{attribute 'linkalways'} 
{attribute 'no_explicit_call' := 'This FB is a CLASS and must be accessed using methods or properties'}
{attribute 'enable_dynamic_creation'}
FUNCTION_BLOCK Node_F_VN_TransformIntoDisplayableImageExp EXTENDS VisionNode
VAR
    ipSrcImage : _ITcVnImage;
    ipDestImage : _ITcVnDisplayableImage;
    bAllowDeepCopy : _BOOL(FALSE);
    hrPrev : _HRESULT(S_OK);
	hresult : _HRESULT(S_OK);
END_VAR

METHOD PUBLIC  Clone : I_Node
VAR
	pNode : POINTER TO Node_F_VN_TransformIntoDisplayableImageExp;
END_VAR
pNode := __NEW(Node_F_VN_TransformIntoDisplayableImageExp);
Clone := pNode^;
END_METHOD

METHOD FB_init : BOOL
VAR_INPUT
	bInitRetains : BOOL; // if TRUE, the retain variables are initialized (warm start / cold start)
	bInCopyCode : BOOL;  // if TRUE, the instance afterwards gets moved into the copy code (online change)
END_VAR
AddInput('ipSrcImage', ipSrcImage);
AddParameter('bAllowDeepCopy', bAllowDeepCopy);
AddInput('hrPrev', hrPrev);
AddOutput('ipDestImage', ipDestImage);
AddOutput('hresult',hresult);
END_METHOD

METHOD PROTECTED OnExecute
hresult.Value := F_VN_TransformIntoDisplayableImageExp(
    ipSrcImage := ipSrcImage.Value,
    bAllowDeepCopy := bAllowDeepCopy.Value,
	ipDestImage := ipDestImage.Value,
	hrPrev:= hrPrev.Value);
END_METHOD

METHOD PUBLIC PreExecutionCheck
VAR_INPUT
	Check : I_PreExecutionChecks;
END_VAR
Check.IsTrue(ipSrcImage.IsValid, 'ipSrcImage must contain an image');
END_METHOD

END_FUNCTION_BLOCK

(* stored: Version 1.1.0.1, ProductVersion 3.1.4024.15
   POU Node_F_VN_TransformIntoDisplayableImageExp: Id {d1cda9be-a710-05ca-1817-66ea43c7cedf}, SpecialFunc None
   Folder Constructor: Id {72e8e653-a9eb-05b6-028f-7be5b22db9a1}
   Method Clone: Id {4f772ea4-47c5-0a4a-267a-73a856c4d11f}
   Method FB_init: Id {456676ca-322a-0cf6-34ce-5a9366bc5071}
   Method OnExecute: Id {be037900-1f0c-08a1-1838-c37d349f3776}
   Method PreExecutionCheck: Id {1becd54c-dd35-0186-310e-20a981ea5248} *)
